FUNCTION_BLOCK SK_MoveNeedleDown (* Skill primitive MoveNeedleDown: Lower the needle to Distance mm below the top; the default is all the way down (parameters: Distance [mm] 0.0..50.0, default 50.0). OPC UA Start(Session, parameters...)/Stop/Abort/Reset(Session) -> [Accepted, ErrorID]; START/HALT/ABORT/RESET from a parent -> SUCCESS or FAILURE(ErrorID) *)
  (* Standard: 61499-2 *)
  (* Version 0.1, 2026-09-28, Project contributors, AAU Smart Production Lab *)
  PACKAGE filler;
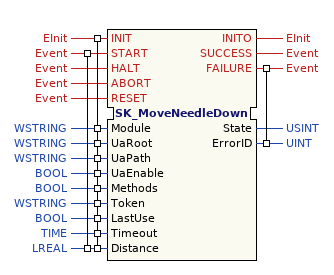
  EVENT_INPUT
    INIT : EInit WITH Module, UaRoot, UaPath, UaEnable, Methods, Token, LastUse, Timeout, Distance;
    START WITH Distance;
    HALT;
    ABORT;
    RESET;
  END_EVENT
  EVENT_OUTPUT
    INITO : EInit;
    SUCCESS;
    FAILURE WITH ErrorID;
  END_EVENT
  VAR_INPUT
    Module : WSTRING;
    UaRoot : WSTRING;
    UaPath : WSTRING;
    UaEnable : BOOL;
    Methods : BOOL;
    Token : WSTRING;
    LastUse : BOOL := TRUE;
    Timeout : TIME := T#5000ms;
    Distance : LREAL := 50.0;
  END_VAR
  VAR_OUTPUT
    State : USINT;
    ErrorID : UINT;
  END_VAR
  (* Group SkillControl: State machine and OPC UA: Start(Session, parameters) with the range check, Stop, Abort, Reset; State, parameters and results published *)
  (* Group Execution: One run: the contract, the command to the equipment and the end condition *)
  (* Group Equipment: The equipment's state in, the command as output values out (the command table and its timed phases are in Driver) *)
  FBS
    Control : modlib::SKILL_Core; {SET_ATTRIBUTE(GroupName, SkillControl)}
    Logic : filler::SL_MoveNeedleDown(Equipment := "NeedleAxis"); {SET_ATTRIBUTE(GroupName, Execution)}
    UaStart : iec61499::net::SERVER_2_2; {SET_ATTRIBUTE(GroupName, SkillControl)}
    Par_Distance : modlib::SKILL_Param_LREAL(Lower := 0.0, Upper := 50.0); {SET_ATTRIBUTE(GroupName, SkillControl)}
    PubParams : iec61499::net::PUBLISH_1; {SET_ATTRIBUTE(GroupName, SkillControl)}
    EqState : iec61499::net::SUBSCRIBE_4(QI := TRUE); {SET_ATTRIBUTE(GroupName, Equipment)}
    EqView : filler::EV_NeedleAxis; {SET_ATTRIBUTE(GroupName, Equipment)}
    WaitT : iec61499::events::E_DELAY(DT := T#500ms); {SET_ATTRIBUTE(GroupName, Execution)}
    Driver : filler::EC_NeedleAxis; {SET_ATTRIBUTE(GroupName, Equipment)}
    PhaseT : iec61499::events::E_DELAY; {SET_ATTRIBUTE(GroupName, Equipment)}
    EqCmd : iec61499::net::PUBLISH_4(QI := TRUE); {SET_ATTRIBUTE(GroupName, Equipment)}
    Timer : iec61499::events::E_DELAY; {SET_ATTRIBUTE(GroupName, Execution)}
  END_FBS
  EVENT_CONNECTIONS
    Control.RSP_START TO UaStart.RSP;
    UaStart.IND TO Par_Distance.CHECK;
    Control.GO TO Par_Distance.LATCH;
    Par_Distance.CHECKED TO Control.CMD_START;
    Par_Distance.LATCHED TO PubParams.REQ;
    PubParams.INITO TO PubParams.REQ;
    INIT TO Control.INIT;
    Control.INITO TO Logic.INIT;
    Logic.INITO TO UaStart.INIT;
    UaStart.INITO TO Par_Distance.INIT;
    Par_Distance.INITO TO PubParams.INIT;
    PubParams.INITO TO EqState.INIT;
    EqState.INITO TO EqCmd.INIT;
    EqCmd.INITO TO INITO;
    START TO Control.START;
    HALT TO Control.HALT;
    ABORT TO Control.ABORT;
    RESET TO Control.RESET;
    Control.SUCCESS TO SUCCESS;
    Control.FAILURE TO FAILURE;
    Par_Distance.LATCHED TO Logic.START;
    Control.HALT_O TO Logic.HALT;
    Control.ABORT_O TO Logic.ABORT;
    Control.RUN_STOP TO Control.STOP_DONE;
    Logic.DONE TO Control.EXEC_DONE;
    Logic.FAILED TO Control.EXEC_FAILED;
    Logic.HALTED TO Control.EXEC_FAILED;
    EqState.IND TO EqView.REQ;
    EqView.CNF TO Logic.SAMPLE;
    Logic.CMD TO Driver.PLAY;
    Driver.OUT TO EqCmd.REQ;
    Driver.PHASE_START TO PhaseT.START;
    Driver.PHASE_STOP TO PhaseT.STOP;
    PhaseT.EO TO Driver.PHASE_T;
    Driver.PLAYED TO Logic.PLAYED;
    Logic.WAIT_START TO WaitT.START;
    Logic.WAIT_STOP TO WaitT.STOP;
    WaitT.EO TO Logic.WAIT_OVER;
    Logic.TIMER_START TO Timer.START;
    Logic.TIMER_STOP TO Timer.STOP;
    Timer.EO TO Logic.TIMER;
  END_CONNECTIONS
  DATA_CONNECTIONS
    Control.IdStart TO UaStart.ID;
    UaStart.RD_1 TO Control.S_Start;
    Control.Accepted TO UaStart.SD_1;
    Control.RspError TO UaStart.SD_2;
    UaStart.RD_2 TO Par_Distance.S;
    Control.FromUa TO Par_Distance.FromUa;
    Par_Distance.P TO PubParams.SD_1;
    Par_Distance.InRange TO Control.InRange;
    Module TO Control.Module;
    UaRoot TO Control.UaRoot;
    UaPath TO Control.UaPath;
    UaEnable TO Control.UaEnable;
    Methods TO Control.Methods;
    Methods TO UaStart.QI;
    Control.State TO State;
    Control.ErrorID TO ErrorID;
    Module TO Logic.Module;
    Token TO Logic.Token;
    LastUse TO Logic.LastUse;
    UaRoot TO Logic.UaRoot;
    UaPath TO Logic.UaPath;
    Timeout TO Logic.Timeout;
    UaEnable TO PubParams.QI;
    Logic.IdParams TO PubParams.ID;
    Distance TO Par_Distance.Default;
    Par_Distance.P TO Logic.Distance;
    Logic.ErrorID TO Control.ExecError;
    Logic.EqFree TO Control.EqFree;
    Logic.IdEqState TO EqState.ID;
    EqState.RD_1 TO EqView.I_AtTop;
    EqState.RD_2 TO EqView.I_AtBottom;
    EqState.RD_3 TO EqView.I_Position;
    EqState.RD_4 TO EqView.I_Holder;
    EqView.AtTop TO Logic.AtTop;
    EqView.AtBottom TO Logic.AtBottom;
    EqView.Position TO Logic.Position;
    EqView.Holder TO Logic.Holder;
    Logic.IdEqCmd TO EqCmd.ID;
    Logic.C_Holder TO Driver.Holder;
    Logic.C_Command TO Driver.Command;
    Logic.C_Release TO Driver.Release;
    Driver.O_Holder TO EqCmd.SD_1;
    Driver.O_Release TO EqCmd.SD_2;
    Driver.N_Down TO EqCmd.SD_3;
    Driver.N_Up TO EqCmd.SD_4;
    Driver.PhaseDT TO PhaseT.DT;
    Logic.TimerDT TO Timer.DT;
  END_CONNECTIONS
END_FUNCTION_BLOCK
